FUNCTION_BLOCK MatrixMulReal_v1 (* Basic FB with empty ECC *)
  (* Standard: 61499-2 *)
  (* Version 1.0, 2020-08-05, Candra Wardaya, UGM *)
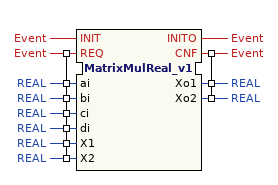
  EVENT_INPUT
    INIT; (* Initialization Input *)
    REQ WITH ai, bi, ci, di, X1, X2; (* Request of Execution *)
  END_EVENT
  EVENT_OUTPUT
    INITO; (* Initialization Output *)
    CNF WITH Xo1, Xo2; (* Confirmation of Execution *)
  END_EVENT
  VAR_INPUT
    ai : REAL; (* Input Matrix Component *)
    bi : REAL; (* Input Matrix Component *)
    ci : REAL; (* Input Matrix Component *)
    di : REAL; (* Input Matrix Component *)
    X1 : REAL; (* Input 2nd Matrix Component *)
    X2 : REAL; (* Input 2nd Matrix Component *)
  END_VAR
  VAR_OUTPUT
    Xo1 : REAL; (* Output 1 *)
    Xo2 : REAL; (* Output 2 *)
  END_VAR
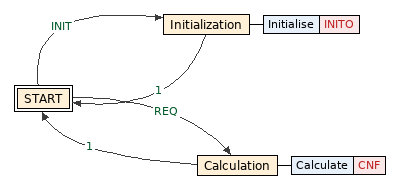
  EC_STATES
    START; (* Initial State *)
    Initialization : Initialise -> INITO;
    Calculation : Calculate -> CNF;
  END_STATES
  EC_TRANSITIONS
    START TO Initialization := INIT;
    Initialization TO START := 1;
    START TO Calculation := REQ;
    Calculation TO START := 1;
  END_TRANSITIONS
  ALGORITHM Initialise IN ST: (* New Algorithm *)

  END_ALGORITHM
  ALGORITHM Calculate IN ST: (* New Algorithm *)
Xo1 := (ai*X1 + bi*X2);
Xo2 := (ci*X1 + di*X2);
  END_ALGORITHM
END_FUNCTION_BLOCK
